// SIMATIC S7-200 SMART project (STEP 7-Micro/WIN SMART), CPU SR40

SYMBOL_TABLE M 符号
急停标志位            M0.0
本地启动标志位          M0.1
远程启动标志位          M0.2
本地停止标志位          M0.3
远程停止标志位          M0.4
主站完成             M1.0
开始读取             M1.1
读取完成1            M1.2
读取完成2            M1.3
读取完成3            M1.4
读取完成4            M1.5
写入完成1            M1.6
写入完成2            M1.7
END_SYMBOL_TABLE

SYMBOL_TABLE 系统符号
Always_On        SM0.0    // 始终接通
First_Scan_On    SM0.1    // 仅在第一个扫描周期时接通
Clock_1s         SM0.5    // 针对 1 s 的周期时间，时钟脉冲接通 0.5 s，断开 0.5 s.
END_SYMBOL_TABLE

SYMBOL_TABLE V 符号
运行指示自动           V10.0
运行指示手动           V10.1
停止指示自动           V10.2
停止指示手动           V10.3
故障指示自动           V10.4
故障指示手动           V10.5
螺杆泵启动自动          V10.6
螺杆泵启动手动          V10.7
罗茨泵启动自动          V11.0
罗茨泵启动手动          V11.1
入口阀自动            V11.2
入口阀手动            V11.3
出口阀自动            V11.4
出口阀手动            V11.5
清洗阀自动            V11.6
清洗阀手动            V11.7
吹扫阀自动            V12.0
吹扫阀手动            V12.1
螺杆泵冷却水阀自动        V12.2
螺杆泵冷却水阀手动        V12.3
罗茨泵冷却水阀自动        V12.4
罗茨泵冷却水阀手动        V12.5
螺杆泵冷却风扇自动        V12.6
螺杆泵冷却风扇手动        V12.7
罗茨泵冷却风扇自动        V13.0
罗茨泵冷却风扇手动        V13.1
排液阀自动            V13.2
排液阀手动            V13.3
罗茨泵启动自动2         V13.4
罗茨泵启动手动2         V13.5
系统故障             V16.0
罗茨泵过载            V16.1
螺杆泵变频器故障报警       V16.2
罗茨泵变频器故障报警       V16.3
冷却水流量低           V16.4
冷却水温度报警          V16.5
冷却水温度停机          V16.6
入口阀打开故障          V16.7
入口阀关闭故障          V17.0
出口阀打开故障          V17.1
出口阀关闭故障          V17.2
螺杆泵冷却风机过载报警      V17.3
罗茨泵冷却风机过载报警      V17.4
螺杆泵维保报警          V17.5
罗茨泵维保报警          V17.6
急停报警             V17.7
罗茨泵变频器故障报警2      V18.0
急停报警2            V18.1
急停报警3            V18.2
运行步              VW20
当前真空度            VD50
当前温度             VD54
排液计时             VW60
清洗计时             VW62
吹扫计时             VW64
冷却水计时            VW66
罗茨泵运行真空度1        VD100
排液间隔时间           VW104
预设清洗时间           VW106
预设吹扫时间           VW108
预设冷却水关闭时间        VW110
螺杆泵手动频率          VW112
罗茨泵手动频率          VW114
螺杆泵停机频率          VW116
冷却水温度报警值         VD118
冷却水温度停机值         VD122
罗茨泵运行真空度2        VD126
罗茨泵停止真空度1        VD130
罗茨泵停止真空度2        VD134
罗茨泵手动频率2         VW138
螺杆泵故障信息          VB200
螺杆泵变频器故障         V201.7
罗茨泵故障信息          VB202
罗茨泵变频器故障         V203.7
罗茨泵故障信息2         VB204
罗茨泵变频器故障2        V205.7
螺杆泵频率电流          VB210
螺杆泵频率            VW210
螺杆泵电流            VW212
罗茨泵频率电流          VB220
罗茨泵频率            VW220
罗茨泵电流            VW222
罗茨泵频率电流2         VB224
罗茨泵频率2           VW224
罗茨泵电流2           VW226
写螺杆泵频率           VB230
螺杆泵频率写入值         VW230
写罗茨泵频率           VB240
罗茨泵频率写入值         VW240
写罗茨泵频率2          VB242
罗茨泵频率写入值2        VW242
中间值1             VD250
中间值2             VD254
螺杆泵当前频率          VD258
中间值3             VD262
中间值4             VD266
螺杆泵当前电流          VD270
中间值5             VD274
中间值6             VD278
罗茨泵当前频率          VD282
中间值7             VD286
中间值8             VD290
罗茨泵当前电流          VD294
写入螺杆泵频率          VW298
写入罗茨泵频率          VW300
写入罗茨泵频率1         VW302
中间值9             VD3000
中间值10            VD3004
中间值11            VD3008
中间值12            VD3012
罗茨泵当前频率2         VD3016
罗茨泵当前电流2         VD3020
写入螺杆泵频率2         VD3024
写入罗茨泵频率2         VD3028
罗茨泵自动频率2         VW3032
中间量13            VW3034
第一页时间1           VW310
第一页时间2           VW312
第一页时间3           VW314
第一页时间4           VW316
第一页时间5           VW318
第一页时间6           VW320
第一页频率1           VW322
第一页频率2           VW324
第一页频率3           VW326
第一页频率4           VW328
第一页频率5           VW330
第一页频率6           VW332
第二页时间1           VW334
第二页时间2           VW336
第二页时间3           VW338
第二页时间4           VW340
第二页时间5           VW342
第二页时间6           VW344
第二页频率1           VW346
第二页频率2           VW348
第二页频率3           VW350
第二页频率4           VW352
第二页频率5           VW354
第二页频率6           VW356
第三页时间1           VW358
第三页时间2           VW360
第三页时间3           VW362
第三页时间4           VW364
第三页时间5           VW366
第三页时间6           VW368
第三页频率1           VW370
第三页频率2           VW372
第三页频率3           VW374
第三页频率4           VW376
第三页频率5           VW378
第三页频率6           VW380
第四页时间1           VW382
第四页时间2           VW384
第四页时间3           VW386
第四页时间4           VW388
第四页时间5           VW390
第四页时间6           VW392
第四页频率1           VW394
第四页频率2           VW396
第四页频率3           VW398
第四页频率4           VW400
第四页频率5           VW402
第四页频率6           VW404
第五页时间1           VW406
第五页时间2           VW408
第五页时间3           VW410
第五页时间4           VW412
第五页时间5           VW414
第五页时间6           VW416
第五页频率1           VW418
第五页频率2           VW420
第五页频率3           VW422
第五页频率4           VW424
第五页频率5           VW426
第五页频率6           VW428
第六页时间1           VW430
第六页时间2           VW432
第六页时间3           VW434
第六页时间4           VW436
第六页时间5           VW438
第六页时间6           VW440
第六页频率1           VW442
第六页频率2           VW444
第六页频率3           VW446
第六页频率4           VW448
第六页频率5           VW450
第六页频率6           VW452
第七页时间1           VW454
第七页时间2           VW456
第七页时间3           VW458
第七页时间4           VW460
第七页时间5           VW462
第七页时间6           VW464
第七页频率1           VW466
第七页频率2           VW468
第七页频率3           VW470
第七页频率4           VW472
第七页频率5           VW474
第七页频率6           VW476
触摸屏页码选择          VW478
实际运行时间1          VW500
实际运行时间2          VW502
实际运行时间3          VW504
实际运行时间4          VW506
实际运行时间5          VW508
实际运行时间6          VW510
实际运行频率1          VW512
实际运行频率2          VW514
实际运行频率3          VW516
实际运行频率4          VW518
实际运行频率5          VW520
实际运行频率6          VW522
step             VW550
螺杆泵自动频率          VW552
罗茨泵自动频率          VW554
螺杆泵运行计时1         VW556
螺杆泵运行计时2         VW558
螺杆泵运行计时3         VW560
螺杆泵运行计时4         VW562
螺杆泵运行计时5         VW564
螺杆泵运行计时6         VW566
中间量9             VW568
螺杆泵总运行时间         VD600
罗茨泵总运行时间         VD604
螺杆泵维保运行时间        VD608
罗茨泵维保运行时间        VD612
螺杆泵维保时间设置        VD616
罗茨泵维保时间设置        VD620
运行时间显示1          VD650    // 螺杆总
运行时间显示2          VD654    // 罗茨总
运行时间显示3          VD658    // 螺杆维保
运行时间显示4          VD662    // 罗茨维保
每秒累加频率1          VD820
每秒累加频率2          VD824
每秒累加频率3          VD828
每秒累加频率4          VD832
每秒累加频率5          VD836
每秒累加频率6          VD840
目标真空度1           VD900
目标真空度2           VD904
目标真空度3           VD908
目标真空度4           VD912
目标真空度5           VD916
目标真空度6           VD920
真空度中间量1          VD924
真空度中间量2          VD928
真空度中间量3          VD932
真空度中间量4          VD936
真空度中间量5          VD940
真空度中间量6          VD944
END_SYMBOL_TABLE

ORGANIZATION_BLOCK MAIN:OB1
TITLE=程序注释
BEGIN
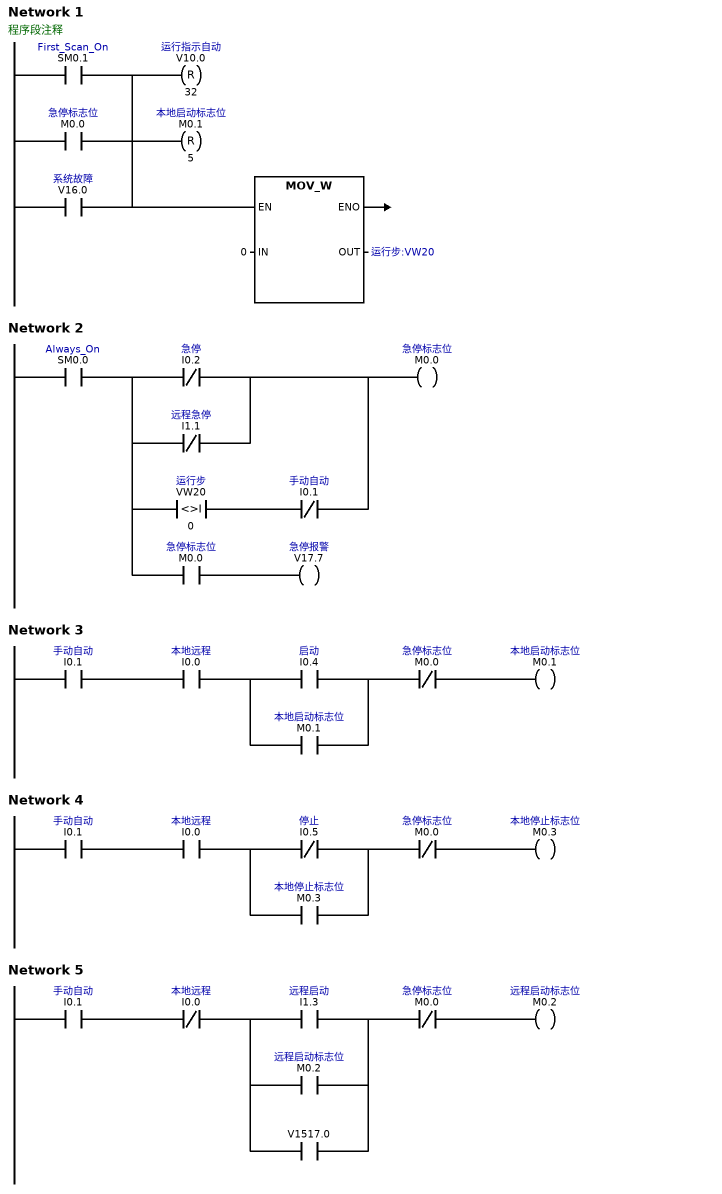
Network 1
// 程序段注释
LD     First_Scan_On:SM0.1
O      急停标志位:M0.0
O      系统故障:V16.0
R      运行指示自动:V10.0, 32
R      本地启动标志位:M0.1, 5
MOVW   0, 运行步:VW20
Network 2
LD     Always_On:SM0.0
LPS
LDN    急停:I0.2
ON     远程急停:I1.1
LDW<>  运行步:VW20, 0
AN     手动自动:I0.1
OLD
ALD
=      急停标志位:M0.0
LPP
A      急停标志位:M0.0
=      急停报警:V17.7
Network 3
LD     手动自动:I0.1
A      本地远程:I0.0
LD     启动:I0.4
O      本地启动标志位:M0.1
ALD
AN     急停标志位:M0.0
=      本地启动标志位:M0.1
Network 4
LD     手动自动:I0.1
A      本地远程:I0.0
LDN    停止:I0.5
O      本地停止标志位:M0.3
ALD
AN     急停标志位:M0.0
=      本地停止标志位:M0.3
Network 5
LD     手动自动:I0.1
AN     本地远程:I0.0
LD     远程启动:I1.3
O      远程启动标志位:M0.2
O      V1517.0
ALD
AN     急停标志位:M0.0
=      远程启动标志位:M0.2
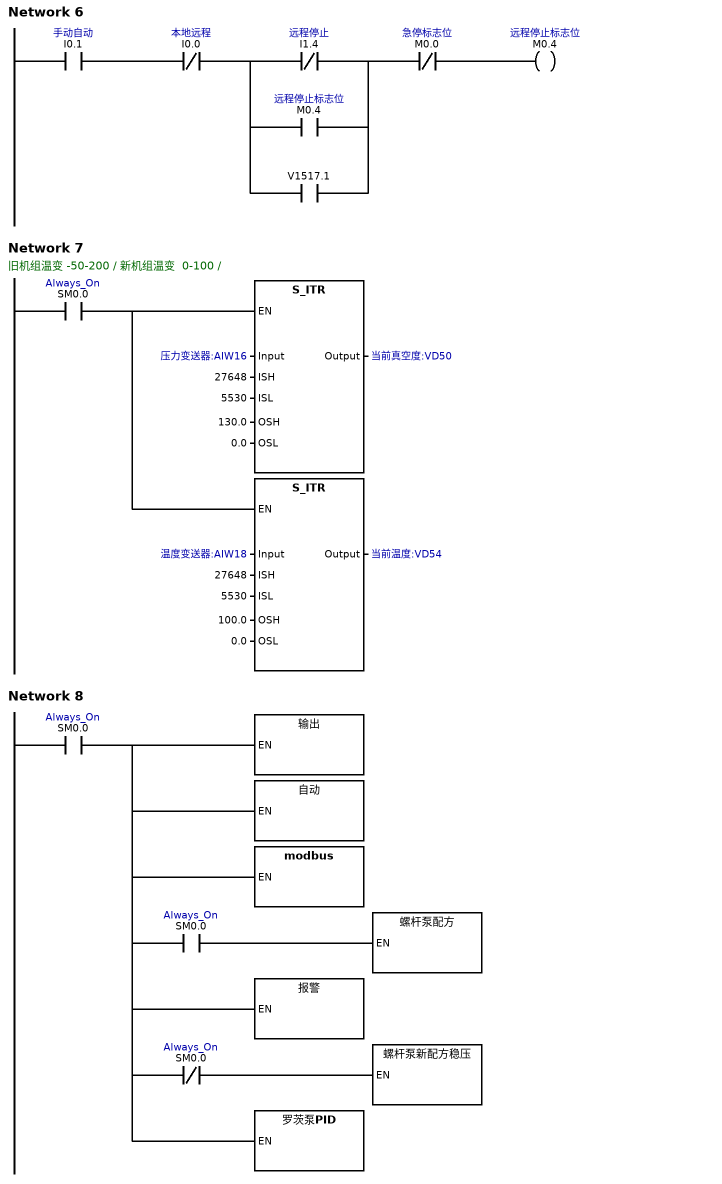
Network 6
LD     手动自动:I0.1
AN     本地远程:I0.0
LDN    远程停止:I1.4
O      远程停止标志位:M0.4
O      V1517.1
ALD
AN     急停标志位:M0.0
=      远程停止标志位:M0.4
Network 7
// 旧机组温变 -50-200
// 新机组温变  0-100
// 
LD     Always_On:SM0.0
CALL   S_ITR:SBR1, 压力变送器:AIW16, 27648, 5530, 130.0, 0.0, 当前真空度:VD50
CALL   S_ITR:SBR1, 温度变送器:AIW18, 27648, 5530, 100.0, 0.0, 当前温度:VD54
Network 8
LD     Always_On:SM0.0
LPS
CALL   输出:SBR0
CALL   自动:SBR2
CALL   modbus:SBR3
A      Always_On:SM0.0
CALL   螺杆泵配方:SBR4
LRD
CALL   报警:SBR6
LRD
AN     Always_On:SM0.0
CALL   螺杆泵新配方稳压:SBR15
LPP
CALL   罗茨泵PID:SBR5
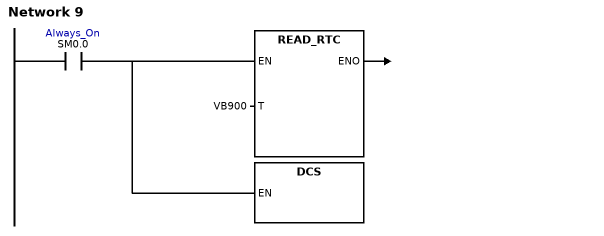
Network 9
LD     Always_On:SM0.0
TODR   VB900
CALL   DCS:SBR11
END_ORGANIZATION_BLOCK

SUBROUTINE_BLOCK 输出:SBR0
TITLE=子程序注释
BEGIN
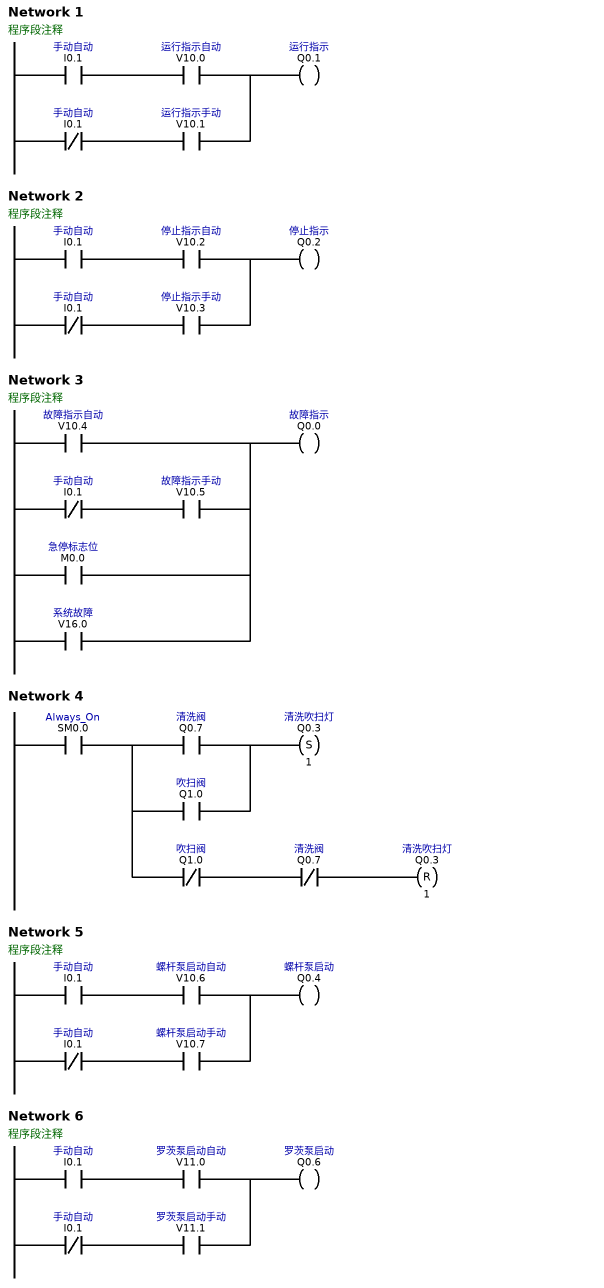
Network 1
// 程序段注释
LD     手动自动:I0.1
A      运行指示自动:V10.0
LDN    手动自动:I0.1
A      运行指示手动:V10.1
OLD
=      运行指示:Q0.1
Network 2
// 程序段注释
LD     手动自动:I0.1
A      停止指示自动:V10.2
LDN    手动自动:I0.1
A      停止指示手动:V10.3
OLD
=      停止指示:Q0.2
Network 3
// 程序段注释
LD     故障指示自动:V10.4
LDN    手动自动:I0.1
A      故障指示手动:V10.5
OLD
O      急停标志位:M0.0
O      系统故障:V16.0
=      故障指示:Q0.0
Network 4
LD     Always_On:SM0.0
LPS
LD     清洗阀:Q0.7
O      吹扫阀:Q1.0
ALD
S      清洗吹扫灯:Q0.3, 1
LPP
AN     吹扫阀:Q1.0
AN     清洗阀:Q0.7
R      清洗吹扫灯:Q0.3, 1
Network 5
// 程序段注释
LD     手动自动:I0.1
A      螺杆泵启动自动:V10.6
LDN    手动自动:I0.1
A      螺杆泵启动手动:V10.7
OLD
=      螺杆泵启动:Q0.4
Network 6
// 程序段注释
LD     手动自动:I0.1
A      罗茨泵启动自动:V11.0
LDN    手动自动:I0.1
A      罗茨泵启动手动:V11.1
OLD
=      罗茨泵启动:Q0.6
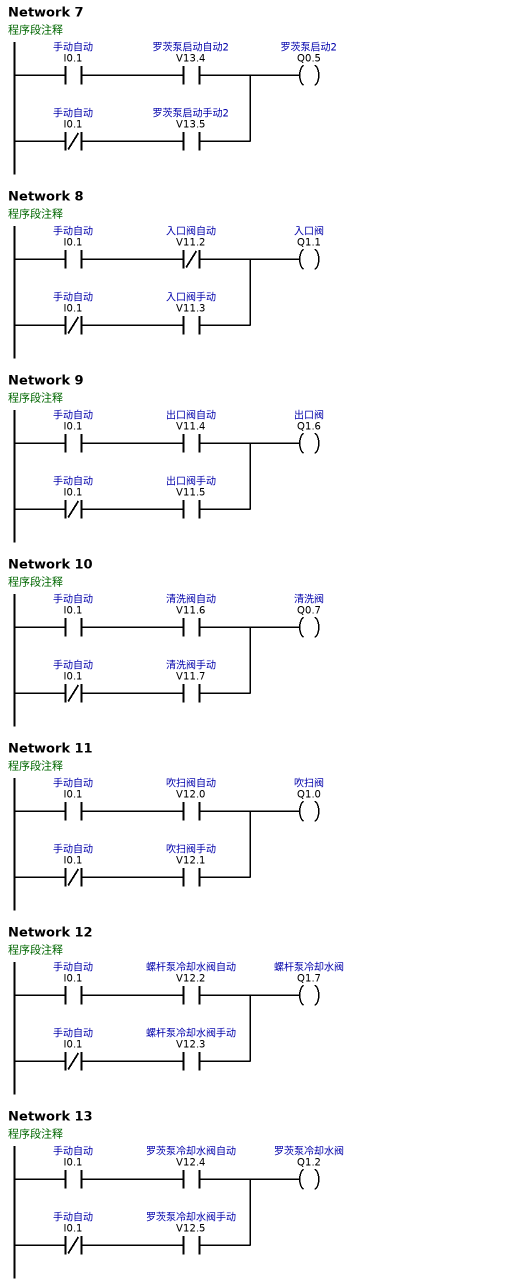
Network 7
// 程序段注释
LD     手动自动:I0.1
A      罗茨泵启动自动2:V13.4
LDN    手动自动:I0.1
A      罗茨泵启动手动2:V13.5
OLD
=      罗茨泵启动2:Q0.5
Network 8
// 程序段注释
LD     手动自动:I0.1
AN     入口阀自动:V11.2
LDN    手动自动:I0.1
A      入口阀手动:V11.3
OLD
=      入口阀:Q1.1
Network 9
// 程序段注释
LD     手动自动:I0.1
A      出口阀自动:V11.4
LDN    手动自动:I0.1
A      出口阀手动:V11.5
OLD
=      出口阀:Q1.6
Network 10
// 程序段注释
LD     手动自动:I0.1
A      清洗阀自动:V11.6
LDN    手动自动:I0.1
A      清洗阀手动:V11.7
OLD
=      清洗阀:Q0.7
Network 11
// 程序段注释
LD     手动自动:I0.1
A      吹扫阀自动:V12.0
LDN    手动自动:I0.1
A      吹扫阀手动:V12.1
OLD
=      吹扫阀:Q1.0
Network 12
// 程序段注释
LD     手动自动:I0.1
A      螺杆泵冷却水阀自动:V12.2
LDN    手动自动:I0.1
A      螺杆泵冷却水阀手动:V12.3
OLD
=      螺杆泵冷却水阀:Q1.7
Network 13
// 程序段注释
LD     手动自动:I0.1
A      罗茨泵冷却水阀自动:V12.4
LDN    手动自动:I0.1
A      罗茨泵冷却水阀手动:V12.5
OLD
=      罗茨泵冷却水阀:Q1.2
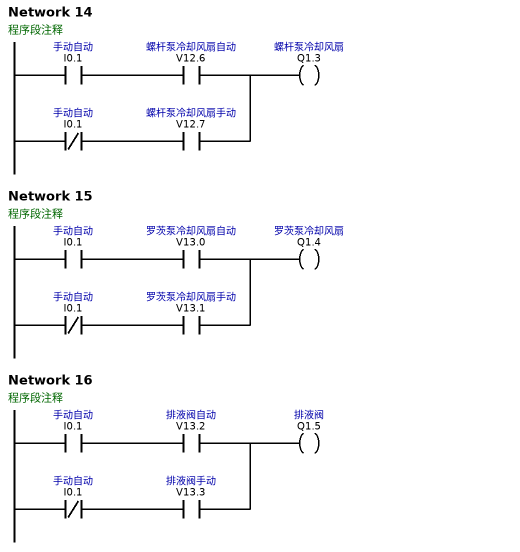
Network 14
// 程序段注释
LD     手动自动:I0.1
A      螺杆泵冷却风扇自动:V12.6
LDN    手动自动:I0.1
A      螺杆泵冷却风扇手动:V12.7
OLD
=      螺杆泵冷却风扇:Q1.3
Network 15
// 程序段注释
LD     手动自动:I0.1
A      罗茨泵冷却风扇自动:V13.0
LDN    手动自动:I0.1
A      罗茨泵冷却风扇手动:V13.1
OLD
=      罗茨泵冷却风扇:Q1.4
Network 16
// 程序段注释
LD     手动自动:I0.1
A      排液阀自动:V13.2
LDN    手动自动:I0.1
A      排液阀手动:V13.3
OLD
=      排液阀:Q1.5
END_SUBROUTINE_BLOCK

// SBR1: protected block, not included

SUBROUTINE_BLOCK 自动:SBR2
TITLE=子程序注释
BEGIN
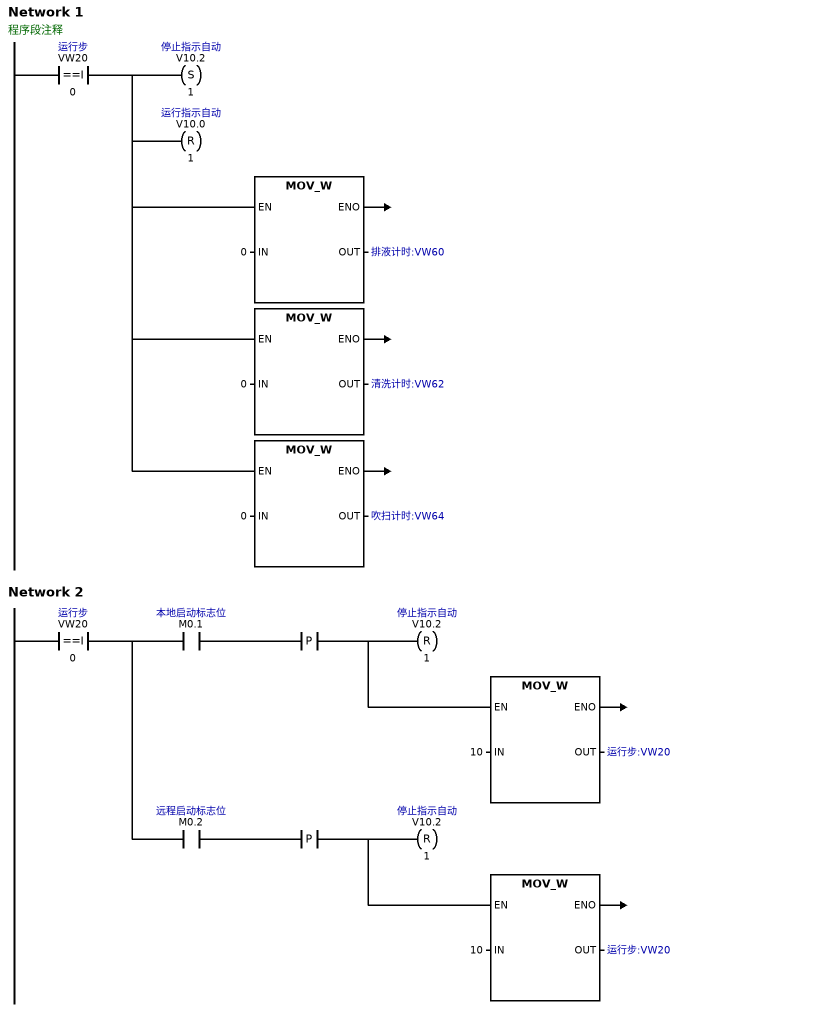
Network 1
// 程序段注释
LDW=   运行步:VW20, 0
S      停止指示自动:V10.2, 1
R      运行指示自动:V10.0, 1
MOVW   0, 排液计时:VW60
MOVW   0, 清洗计时:VW62
MOVW   0, 吹扫计时:VW64
Network 2
LDW=   运行步:VW20, 0
LPS
A      本地启动标志位:M0.1
EU
R      停止指示自动:V10.2, 1
MOVW   10, 运行步:VW20
LPP
A      远程启动标志位:M0.2
EU
R      停止指示自动:V10.2, 1
MOVW   10, 运行步:VW20
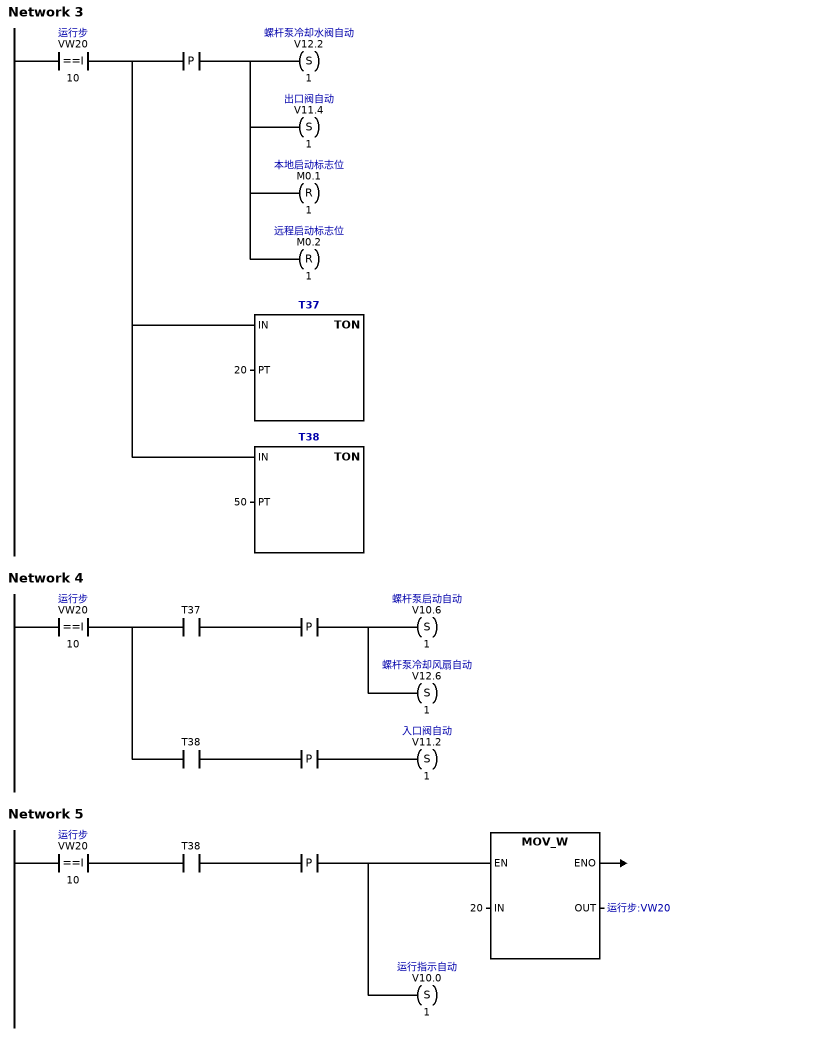
Network 3
LDW=   运行步:VW20, 10
LPS
EU
S      螺杆泵冷却水阀自动:V12.2, 1
S      出口阀自动:V11.4, 1
R      本地启动标志位:M0.1, 1
R      远程启动标志位:M0.2, 1
LPP
TON    T37, 20
TON    T38, 50
Network 4
LDW=   运行步:VW20, 10
LPS
A      T37
EU
S      螺杆泵启动自动:V10.6, 1
S      螺杆泵冷却风扇自动:V12.6, 1
LPP
A      T38
EU
S      入口阀自动:V11.2, 1
Network 5
LDW=   运行步:VW20, 10
A      T38
EU
MOVW   20, 运行步:VW20
S      运行指示自动:V10.0, 1
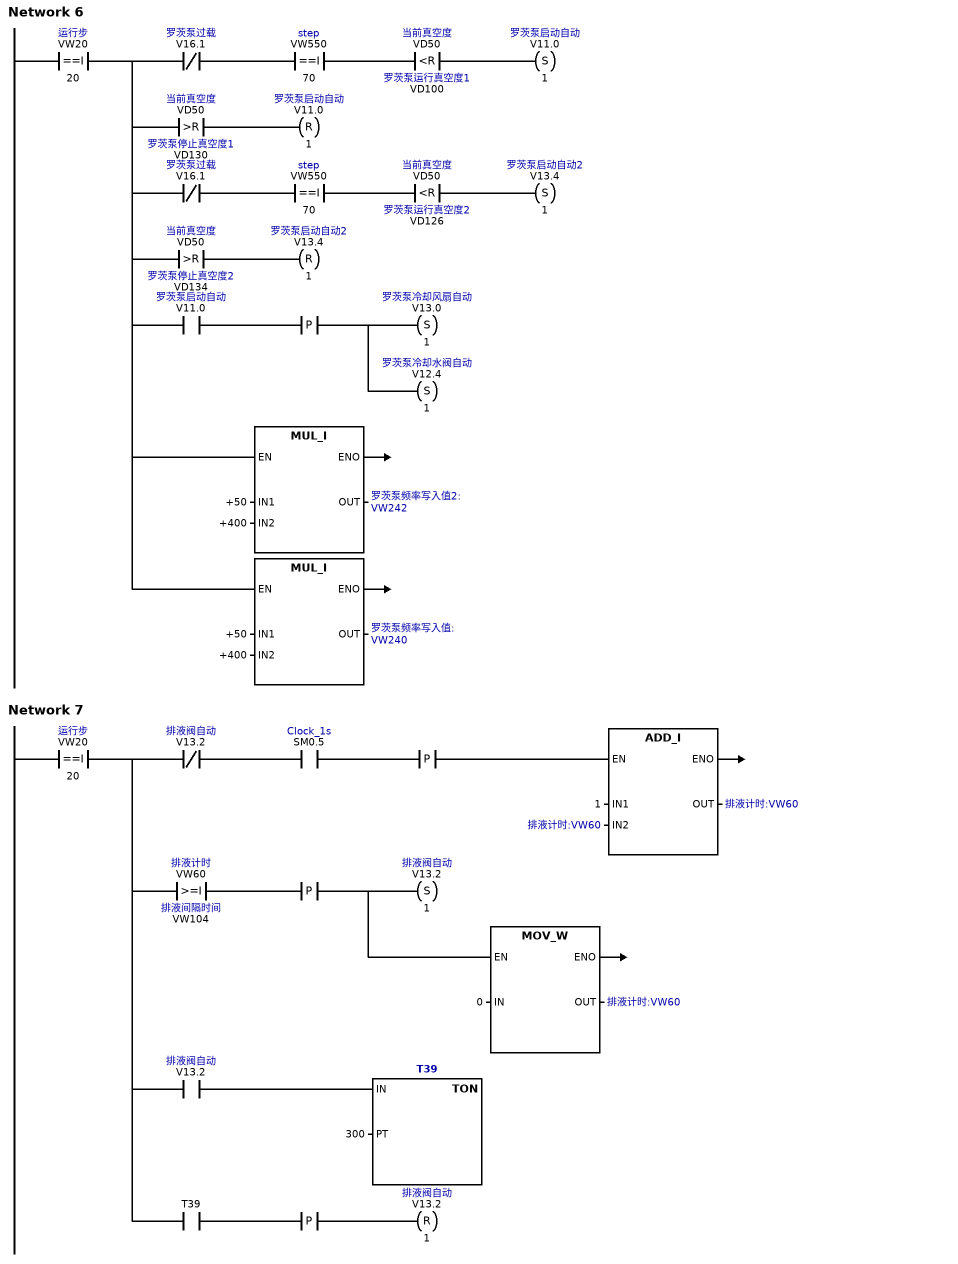
Network 6
LDW=   运行步:VW20, 20
LPS
AN     罗茨泵过载:V16.1
AW=    step:VW550, 70
AR<    当前真空度:VD50, 罗茨泵运行真空度1:VD100
S      罗茨泵启动自动:V11.0, 1
LRD
AR>    当前真空度:VD50, 罗茨泵停止真空度1:VD130
R      罗茨泵启动自动:V11.0, 1
LRD
AN     罗茨泵过载:V16.1
AW=    step:VW550, 70
AR<    当前真空度:VD50, 罗茨泵运行真空度2:VD126
S      罗茨泵启动自动2:V13.4, 1
LRD
AR>    当前真空度:VD50, 罗茨泵停止真空度2:VD134
R      罗茨泵启动自动2:V13.4, 1
LRD
A      罗茨泵启动自动:V11.0
EU
S      罗茨泵冷却风扇自动:V13.0, 1
S      罗茨泵冷却水阀自动:V12.4, 1
LPP
MOVW   +50, 罗茨泵频率写入值2:VW242
*I     +400, 罗茨泵频率写入值2:VW242
MOVW   +50, 罗茨泵频率写入值:VW240
*I     +400, 罗茨泵频率写入值:VW240
Network 7
LDW=   运行步:VW20, 20
LPS
AN     排液阀自动:V13.2
A      Clock_1s:SM0.5
EU
+I     1, 排液计时:VW60
LRD
AW>=   排液计时:VW60, 排液间隔时间:VW104
EU
S      排液阀自动:V13.2, 1
MOVW   0, 排液计时:VW60
LPP
LPS
A      排液阀自动:V13.2
TON    T39, 300
LPP
A      T39
EU
R      排液阀自动:V13.2, 1
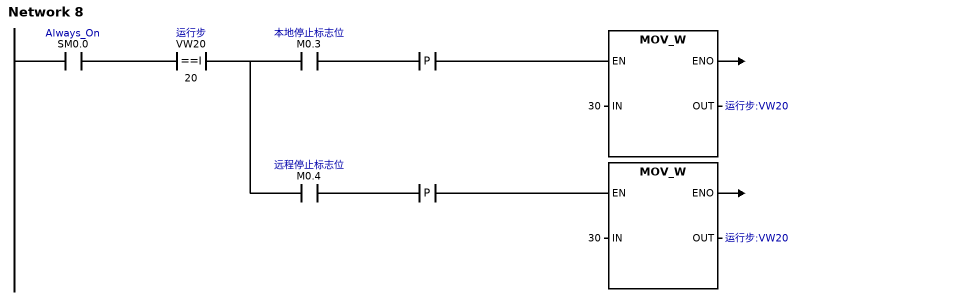
Network 8
LD     Always_On:SM0.0
AW=    运行步:VW20, 20
LPS
A      本地停止标志位:M0.3
EU
MOVW   30, 运行步:VW20
LPP
A      远程停止标志位:M0.4
EU
MOVW   30, 运行步:VW20
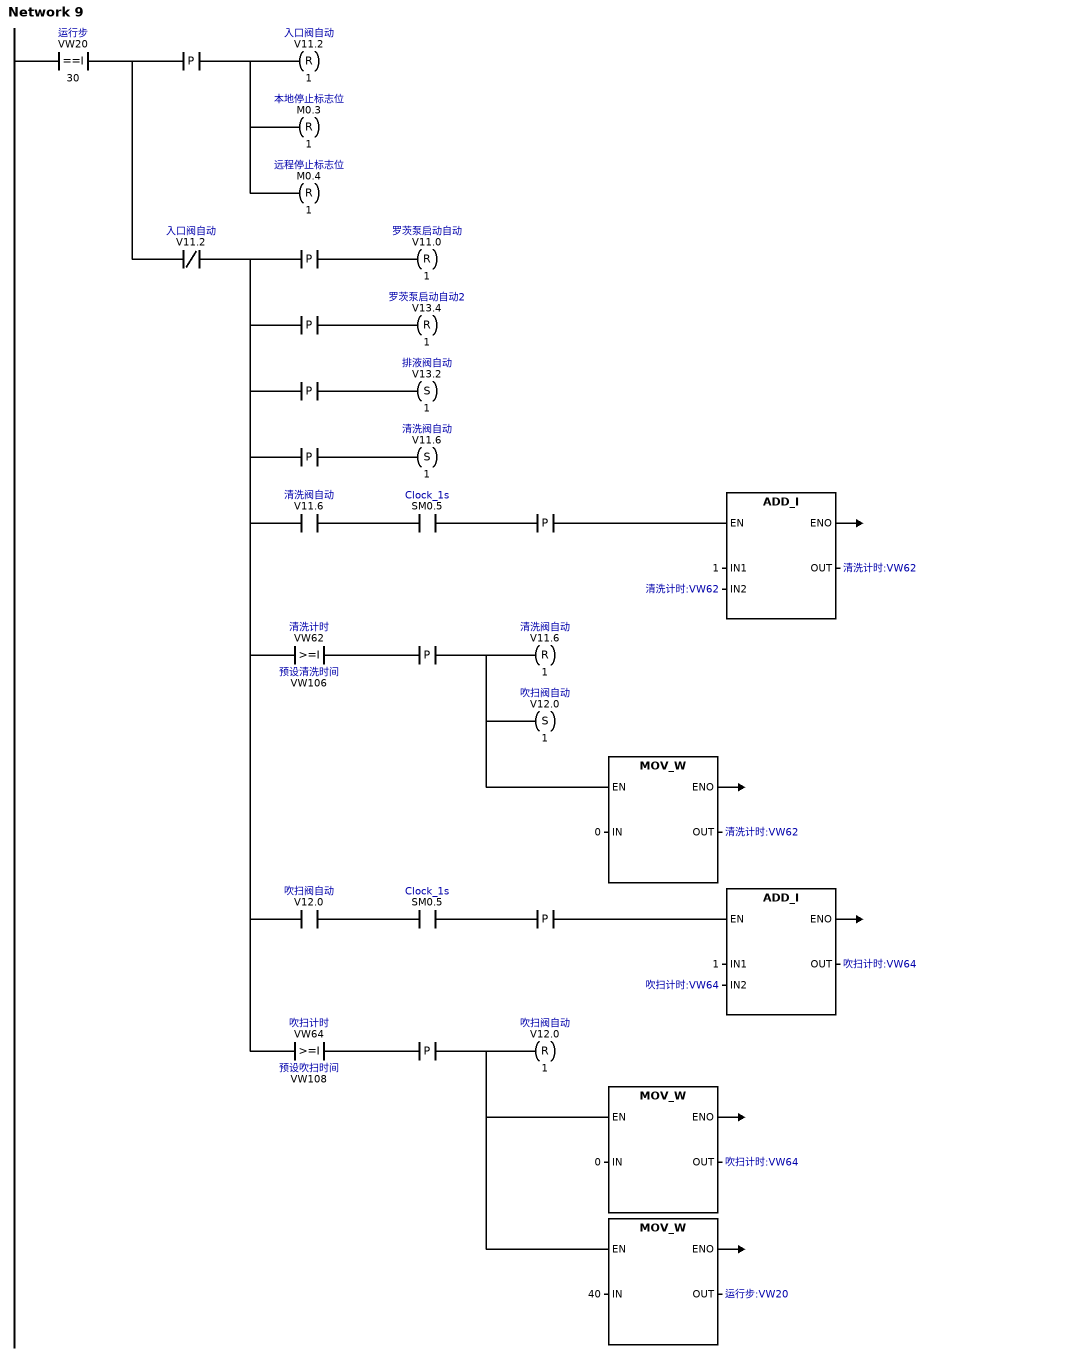
Network 9
LDW=   运行步:VW20, 30
LPS
EU
R      入口阀自动:V11.2, 1
R      本地停止标志位:M0.3, 1
R      远程停止标志位:M0.4, 1
LPP
AN     入口阀自动:V11.2
LPS
EU
R      罗茨泵启动自动:V11.0, 1
LRD
EU
R      罗茨泵启动自动2:V13.4, 1
LRD
EU
S      排液阀自动:V13.2, 1
LRD
EU
S      清洗阀自动:V11.6, 1
LRD
A      清洗阀自动:V11.6
A      Clock_1s:SM0.5
EU
+I     1, 清洗计时:VW62
LRD
AW>=   清洗计时:VW62, 预设清洗时间:VW106
EU
R      清洗阀自动:V11.6, 1
S      吹扫阀自动:V12.0, 1
MOVW   0, 清洗计时:VW62
LRD
A      吹扫阀自动:V12.0
A      Clock_1s:SM0.5
EU
+I     1, 吹扫计时:VW64
LPP
AW>=   吹扫计时:VW64, 预设吹扫时间:VW108
EU
R      吹扫阀自动:V12.0, 1
MOVW   0, 吹扫计时:VW64
MOVW   40, 运行步:VW20
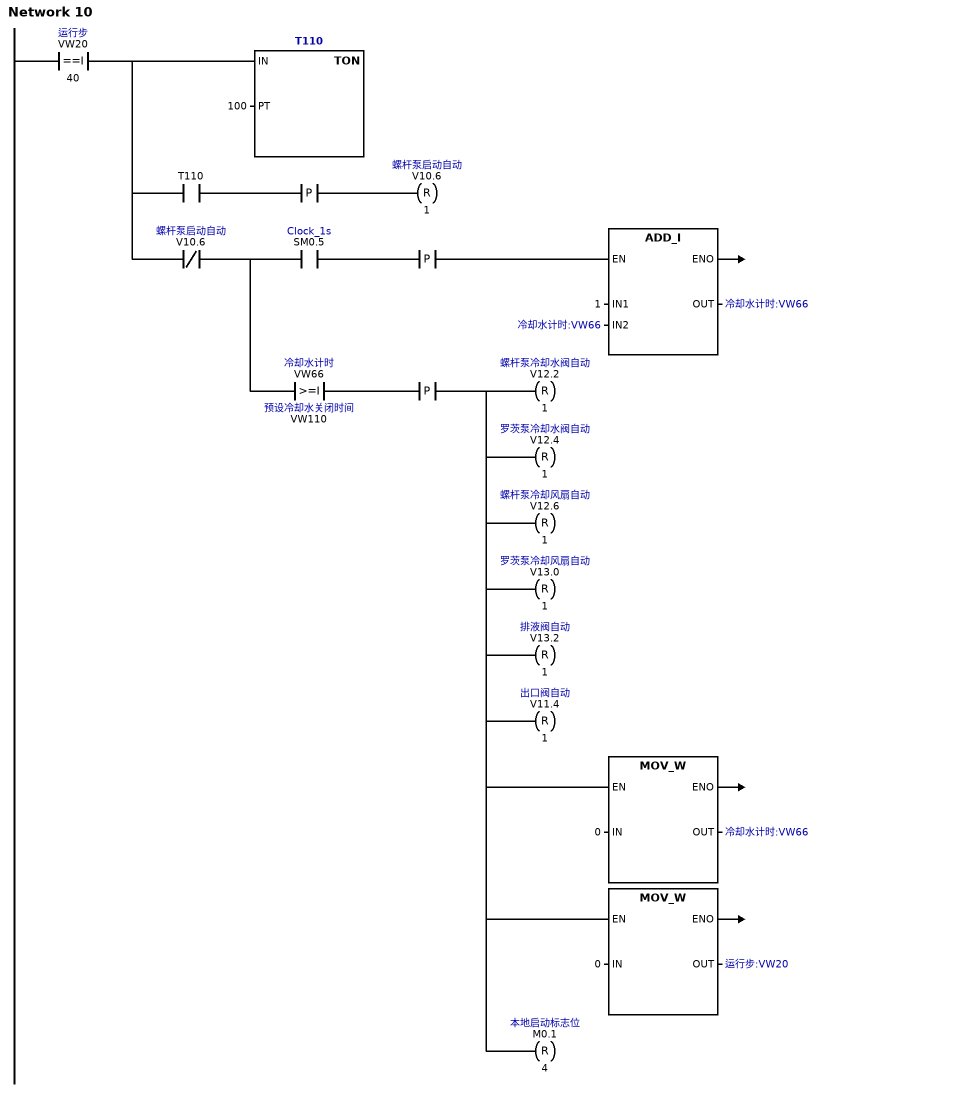
Network 10
LDW=   运行步:VW20, 40
LPS
TON    T110, 100
A      T110
EU
R      螺杆泵启动自动:V10.6, 1
LPP
AN     螺杆泵启动自动:V10.6
LPS
A      Clock_1s:SM0.5
EU
+I     1, 冷却水计时:VW66
LPP
AW>=   冷却水计时:VW66, 预设冷却水关闭时间:VW110
EU
R      螺杆泵冷却水阀自动:V12.2, 1
R      罗茨泵冷却水阀自动:V12.4, 1
R      螺杆泵冷却风扇自动:V12.6, 1
R      罗茨泵冷却风扇自动:V13.0, 1
R      排液阀自动:V13.2, 1
R      出口阀自动:V11.4, 1
MOVW   0, 冷却水计时:VW66
MOVW   0, 运行步:VW20
R      本地启动标志位:M0.1, 4
END_SUBROUTINE_BLOCK

SUBROUTINE_BLOCK modbus:SBR3
TITLE=子程序注释
BEGIN
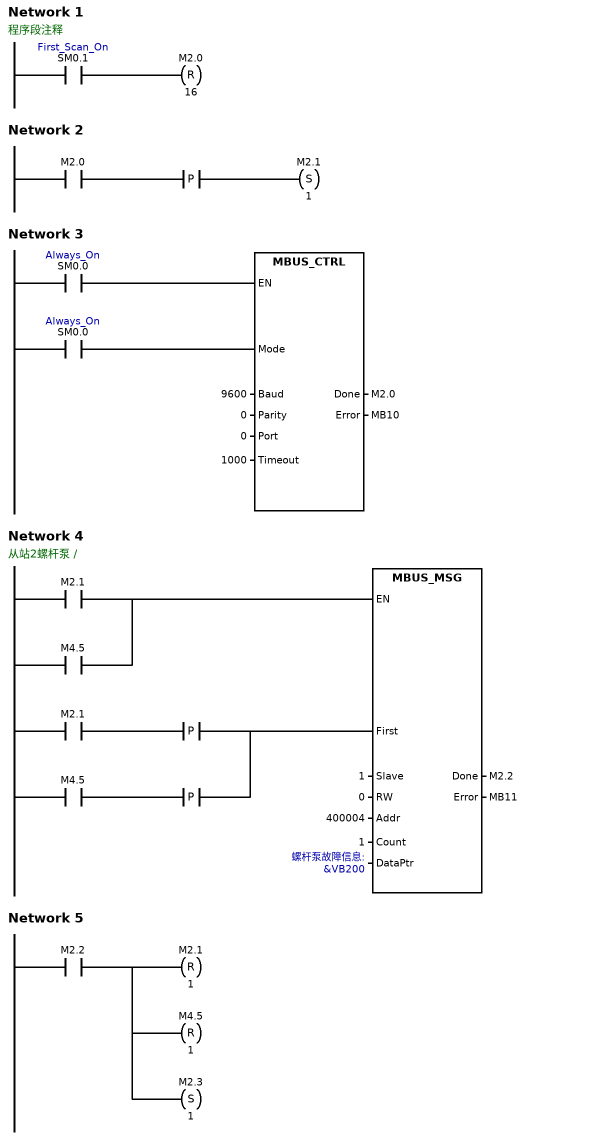
Network 1
// 程序段注释
LD     First_Scan_On:SM0.1
R      M2.0, 16
Network 2
LD     M2.0
EU
S      M2.1, 1
Network 3
LD     Always_On:SM0.0
=      L60.0
LD     Always_On:SM0.0
=      L63.7
LD     L60.0
CALL   MBUS_CTRL:SBR7, L63.7, 9600, 0, 0, 1000, M2.0, MB10
Network 4
// 从站2螺杆泵
// 
LD     M2.1
O      M4.5
=      L60.0
LD     M2.1
EU
LD     M4.5
EU
OLD
=      L63.7
LD     L60.0
CALL   MBUS_MSG:SBR8, L63.7, 1, 0, 400004, 1, &螺杆泵故障信息:VB200, M2.2, MB11
Network 5
LD     M2.2
R      M2.1, 1
R      M4.5, 1
S      M2.3, 1
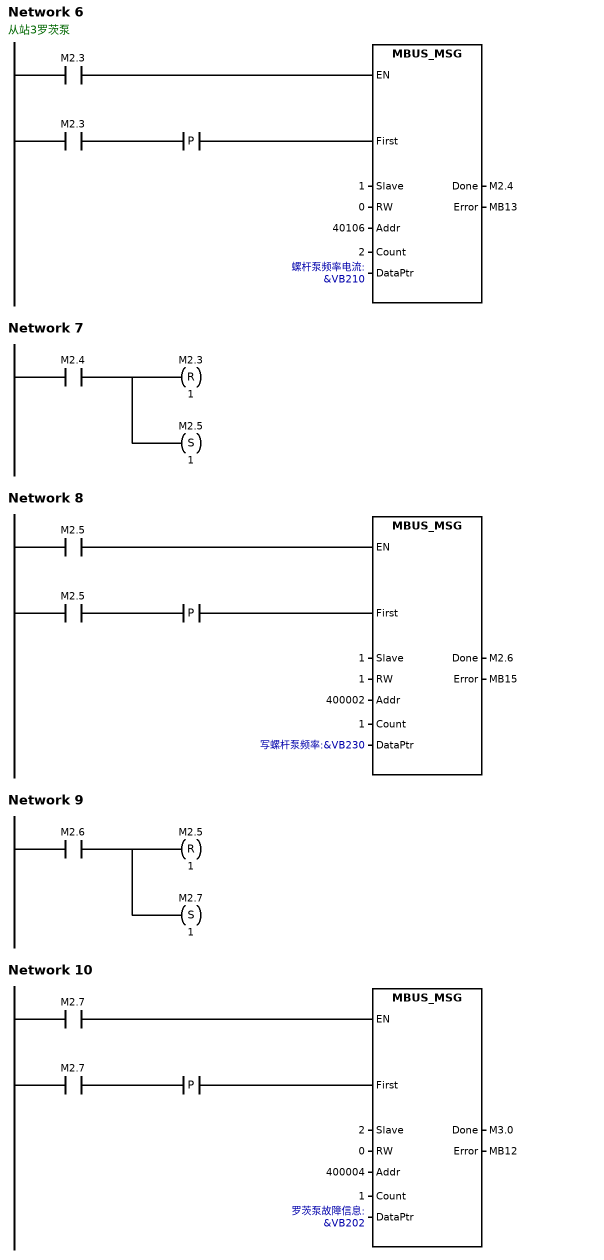
Network 6
// 从站3罗茨泵
LD     M2.3
=      L60.0
LD     M2.3
EU
=      L63.7
LD     L60.0
CALL   MBUS_MSG:SBR8, L63.7, 1, 0, 40106, 2, &螺杆泵频率电流:VB210, M2.4, MB13
Network 7
LD     M2.4
R      M2.3, 1
S      M2.5, 1
Network 8
LD     M2.5
=      L60.0
LD     M2.5
EU
=      L63.7
LD     L60.0
CALL   MBUS_MSG:SBR8, L63.7, 1, 1, 400002, 1, &写螺杆泵频率:VB230, M2.6, MB15
Network 9
LD     M2.6
R      M2.5, 1
S      M2.7, 1
Network 10
LD     M2.7
=      L60.0
LD     M2.7
EU
=      L63.7
LD     L60.0
CALL   MBUS_MSG:SBR8, L63.7, 2, 0, 400004, 1, &罗茨泵故障信息:VB202, M3.0, MB12
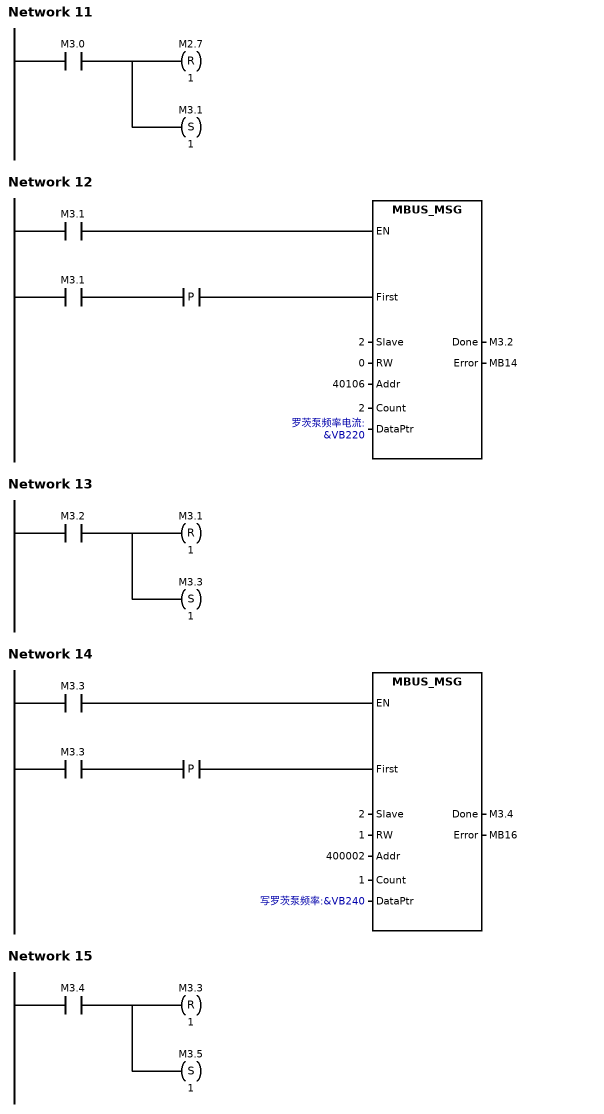
Network 11
LD     M3.0
R      M2.7, 1
S      M3.1, 1
Network 12
LD     M3.1
=      L60.0
LD     M3.1
EU
=      L63.7
LD     L60.0
CALL   MBUS_MSG:SBR8, L63.7, 2, 0, 40106, 2, &罗茨泵频率电流:VB220, M3.2, MB14
Network 13
LD     M3.2
R      M3.1, 1
S      M3.3, 1
Network 14
LD     M3.3
=      L60.0
LD     M3.3
EU
=      L63.7
LD     L60.0
CALL   MBUS_MSG:SBR8, L63.7, 2, 1, 400002, 1, &写罗茨泵频率:VB240, M3.4, MB16
Network 15
LD     M3.4
R      M3.3, 1
S      M3.5, 1
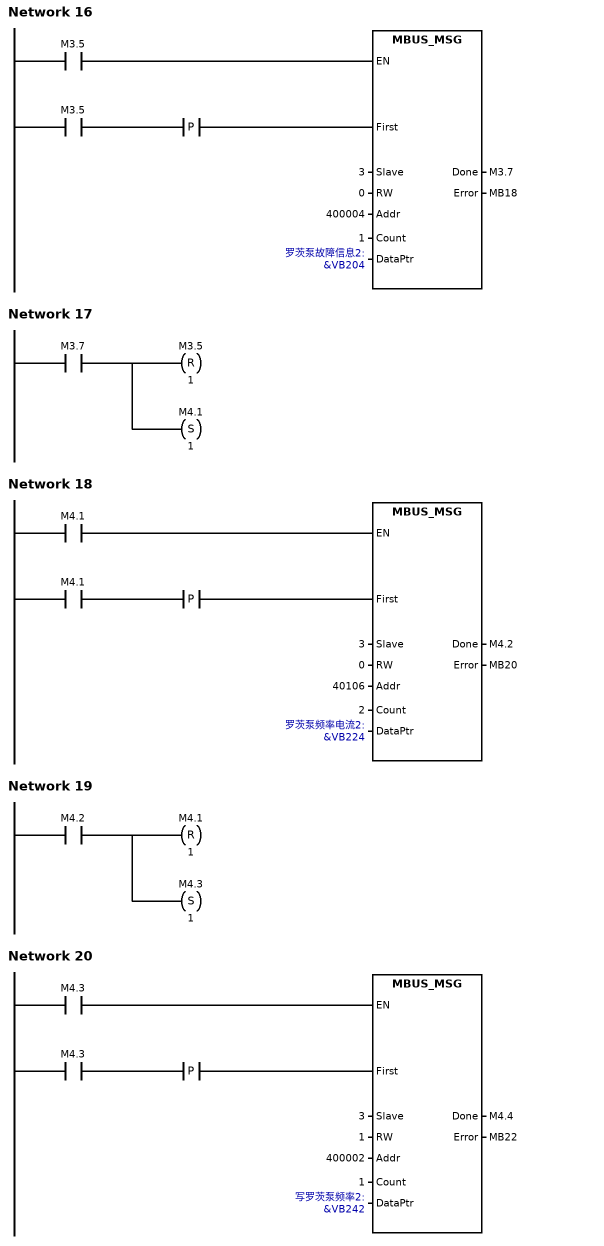
Network 16
LD     M3.5
=      L60.0
LD     M3.5
EU
=      L63.7
LD     L60.0
CALL   MBUS_MSG:SBR8, L63.7, 3, 0, 400004, 1, &罗茨泵故障信息2:VB204, M3.7, MB18
Network 17
LD     M3.7
R      M3.5, 1
S      M4.1, 1
Network 18
LD     M4.1
=      L60.0
LD     M4.1
EU
=      L63.7
LD     L60.0
CALL   MBUS_MSG:SBR8, L63.7, 3, 0, 40106, 2, &罗茨泵频率电流2:VB224, M4.2, MB20
Network 19
LD     M4.2
R      M4.1, 1
S      M4.3, 1
Network 20
LD     M4.3
=      L60.0
LD     M4.3
EU
=      L63.7
LD     L60.0
CALL   MBUS_MSG:SBR8, L63.7, 3, 1, 400002, 1, &写罗茨泵频率2:VB242, M4.4, MB22
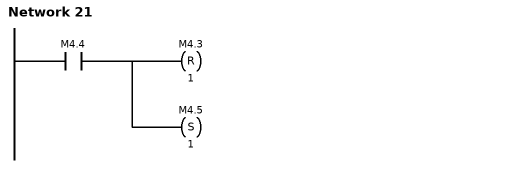
Network 21
LD     M4.4
R      M4.3, 1
S      M4.5, 1
END_SUBROUTINE_BLOCK

SUBROUTINE_BLOCK 螺杆泵配方:SBR4
TITLE=子程序注释
BEGIN
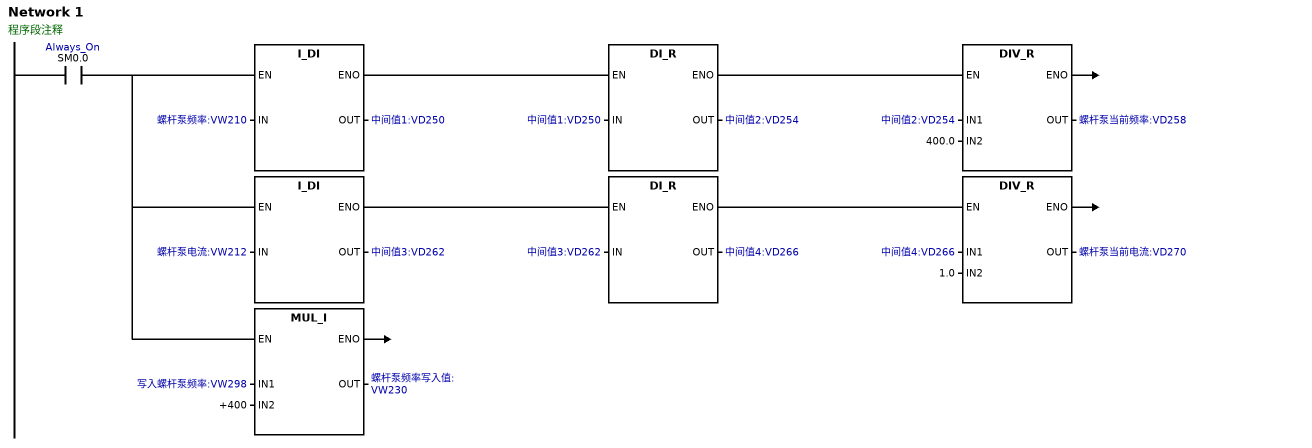
Network 1
// 程序段注释
LD     Always_On:SM0.0
LPS
ITD    螺杆泵频率:VW210, 中间值1:VD250
AENO
DTR    中间值1:VD250, 中间值2:VD254
AENO
MOVR   中间值2:VD254, 螺杆泵当前频率:VD258
/R     400.0, 螺杆泵当前频率:VD258
LRD
ITD    螺杆泵电流:VW212, 中间值3:VD262
AENO
DTR    中间值3:VD262, 中间值4:VD266
AENO
MOVR   中间值4:VD266, 螺杆泵当前电流:VD270
/R     1.0, 螺杆泵当前电流:VD270
LPP
MOVW   写入螺杆泵频率:VW298, 螺杆泵频率写入值:VW230
*I     +400, 螺杆泵频率写入值:VW230
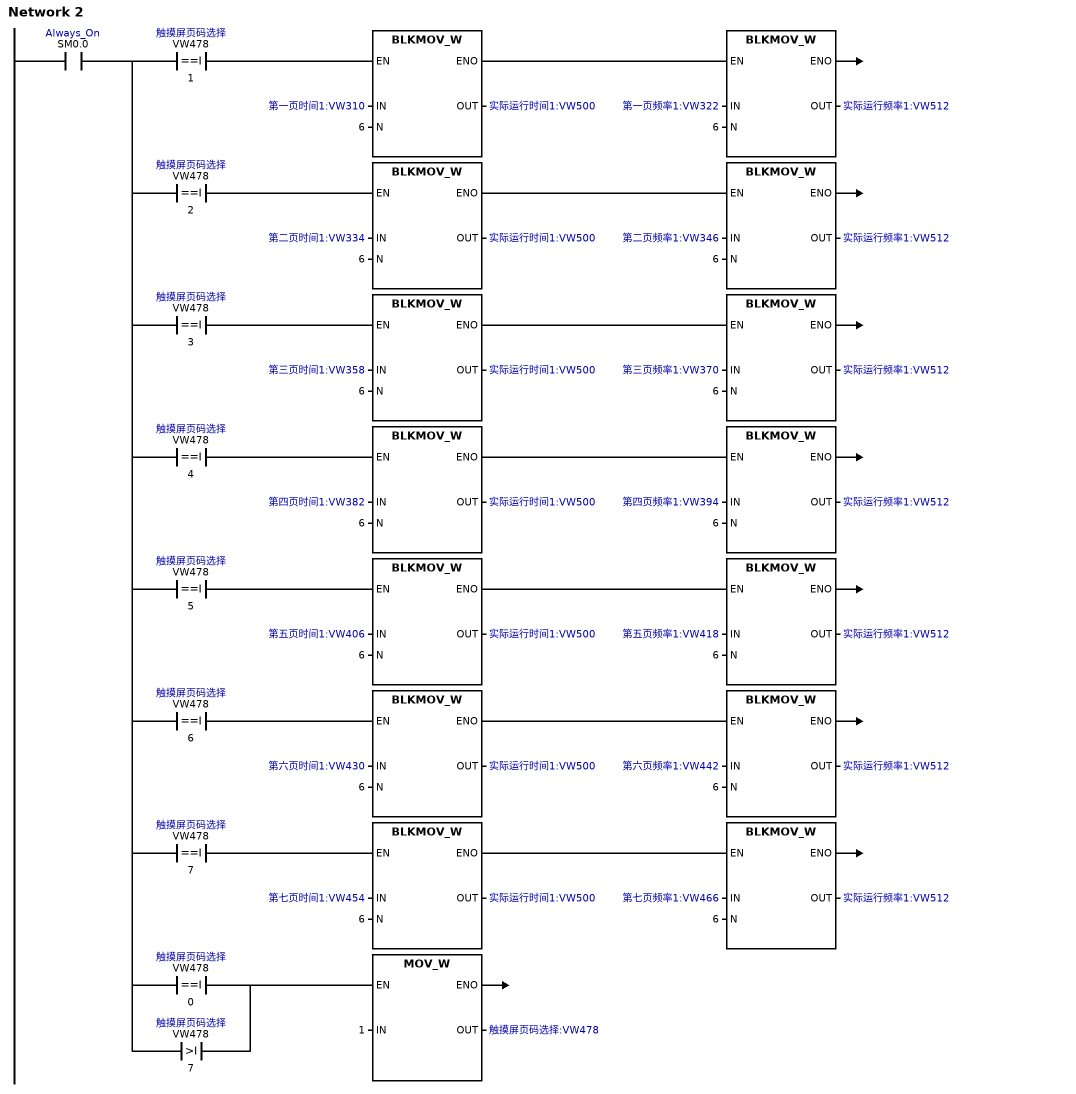
Network 2
LD     Always_On:SM0.0
LPS
AW=    触摸屏页码选择:VW478, 1
BMW    第一页时间1:VW310, 实际运行时间1:VW500, 6
AENO
BMW    第一页频率1:VW322, 实际运行频率1:VW512, 6
LRD
AW=    触摸屏页码选择:VW478, 2
BMW    第二页时间1:VW334, 实际运行时间1:VW500, 6
AENO
BMW    第二页频率1:VW346, 实际运行频率1:VW512, 6
LRD
AW=    触摸屏页码选择:VW478, 3
BMW    第三页时间1:VW358, 实际运行时间1:VW500, 6
AENO
BMW    第三页频率1:VW370, 实际运行频率1:VW512, 6
LRD
AW=    触摸屏页码选择:VW478, 4
BMW    第四页时间1:VW382, 实际运行时间1:VW500, 6
AENO
BMW    第四页频率1:VW394, 实际运行频率1:VW512, 6
LRD
AW=    触摸屏页码选择:VW478, 5
BMW    第五页时间1:VW406, 实际运行时间1:VW500, 6
AENO
BMW    第五页频率1:VW418, 实际运行频率1:VW512, 6
LRD
AW=    触摸屏页码选择:VW478, 6
BMW    第六页时间1:VW430, 实际运行时间1:VW500, 6
AENO
BMW    第六页频率1:VW442, 实际运行频率1:VW512, 6
LRD
AW=    触摸屏页码选择:VW478, 7
BMW    第七页时间1:VW454, 实际运行时间1:VW500, 6
AENO
BMW    第七页频率1:VW466, 实际运行频率1:VW512, 6
LPP
LDW=   触摸屏页码选择:VW478, 0
OW>    触摸屏页码选择:VW478, 7
ALD
MOVW   1, 触摸屏页码选择:VW478
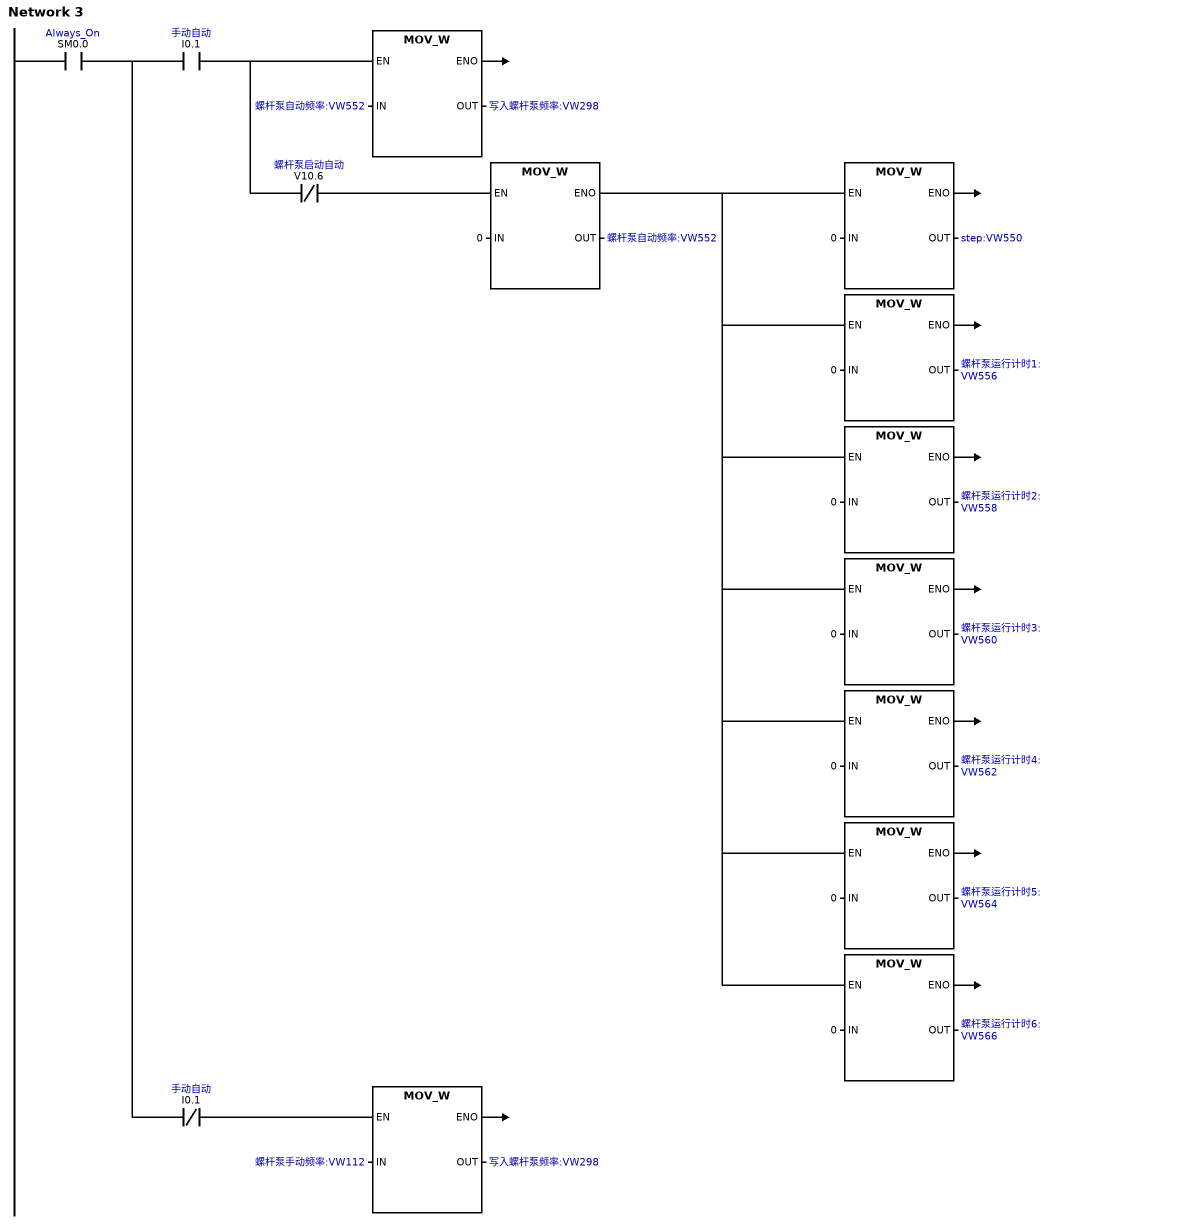
Network 3
LD     Always_On:SM0.0
LPS
A      手动自动:I0.1
MOVW   螺杆泵自动频率:VW552, 写入螺杆泵频率:VW298
AN     螺杆泵启动自动:V10.6
MOVW   0, 螺杆泵自动频率:VW552
AENO
MOVW   0, step:VW550
MOVW   0, 螺杆泵运行计时1:VW556
MOVW   0, 螺杆泵运行计时2:VW558
MOVW   0, 螺杆泵运行计时3:VW560
MOVW   0, 螺杆泵运行计时4:VW562
MOVW   0, 螺杆泵运行计时5:VW564
MOVW   0, 螺杆泵运行计时6:VW566
LPP
AN     手动自动:I0.1
MOVW   螺杆泵手动频率:VW112, 写入螺杆泵频率:VW298
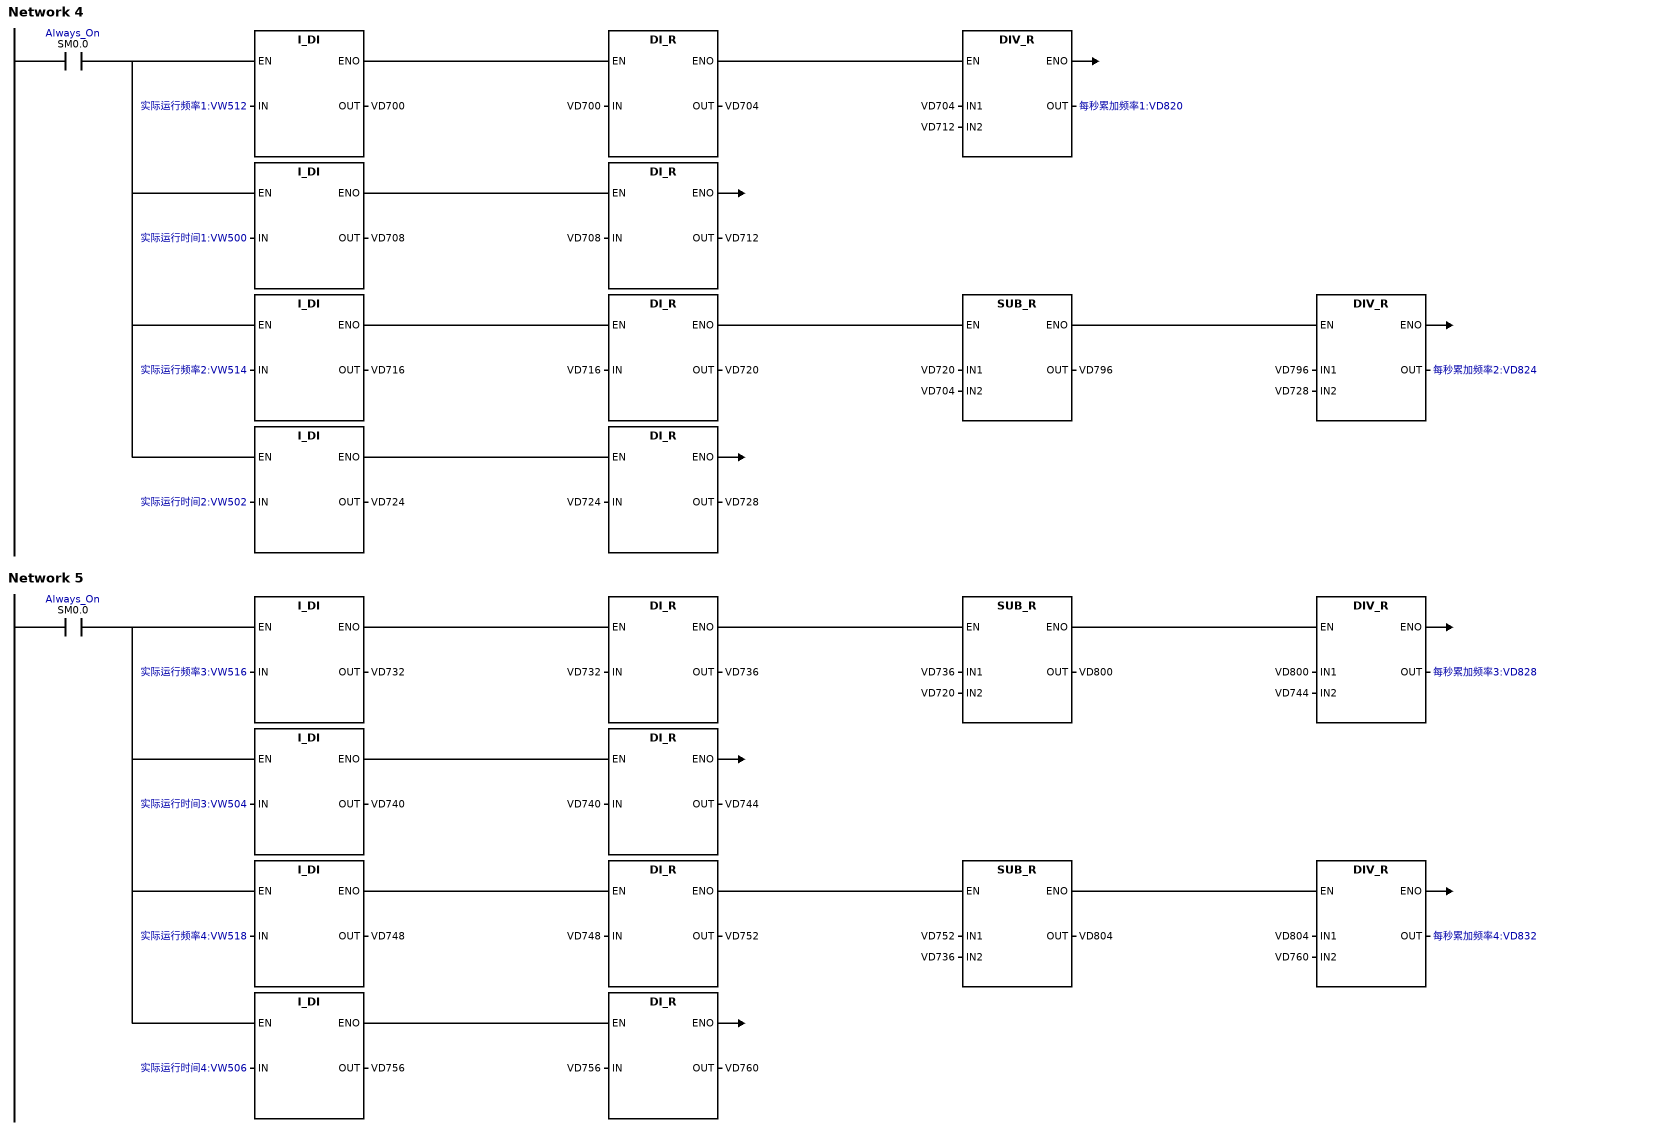
Network 4
LD     Always_On:SM0.0
LPS
ITD    实际运行频率1:VW512, VD700
AENO
DTR    VD700, VD704
AENO
MOVR   VD704, 每秒累加频率1:VD820
/R     VD712, 每秒累加频率1:VD820
LRD
ITD    实际运行时间1:VW500, VD708
AENO
DTR    VD708, VD712
LRD
ITD    实际运行频率2:VW514, VD716
AENO
DTR    VD716, VD720
AENO
MOVR   VD720, VD796
AENO
-R     VD704, VD796
AENO
MOVR   VD796, 每秒累加频率2:VD824
/R     VD728, 每秒累加频率2:VD824
LPP
ITD    实际运行时间2:VW502, VD724
AENO
DTR    VD724, VD728
Network 5
LD     Always_On:SM0.0
LPS
ITD    实际运行频率3:VW516, VD732
AENO
DTR    VD732, VD736
AENO
MOVR   VD736, VD800
AENO
-R     VD720, VD800
AENO
MOVR   VD800, 每秒累加频率3:VD828
/R     VD744, 每秒累加频率3:VD828
LRD
ITD    实际运行时间3:VW504, VD740
AENO
DTR    VD740, VD744
LRD
ITD    实际运行频率4:VW518, VD748
AENO
DTR    VD748, VD752
AENO
MOVR   VD752, VD804
AENO
-R     VD736, VD804
AENO
MOVR   VD804, 每秒累加频率4:VD832
/R     VD760, 每秒累加频率4:VD832
LPP
ITD    实际运行时间4:VW506, VD756
AENO
DTR    VD756, VD760
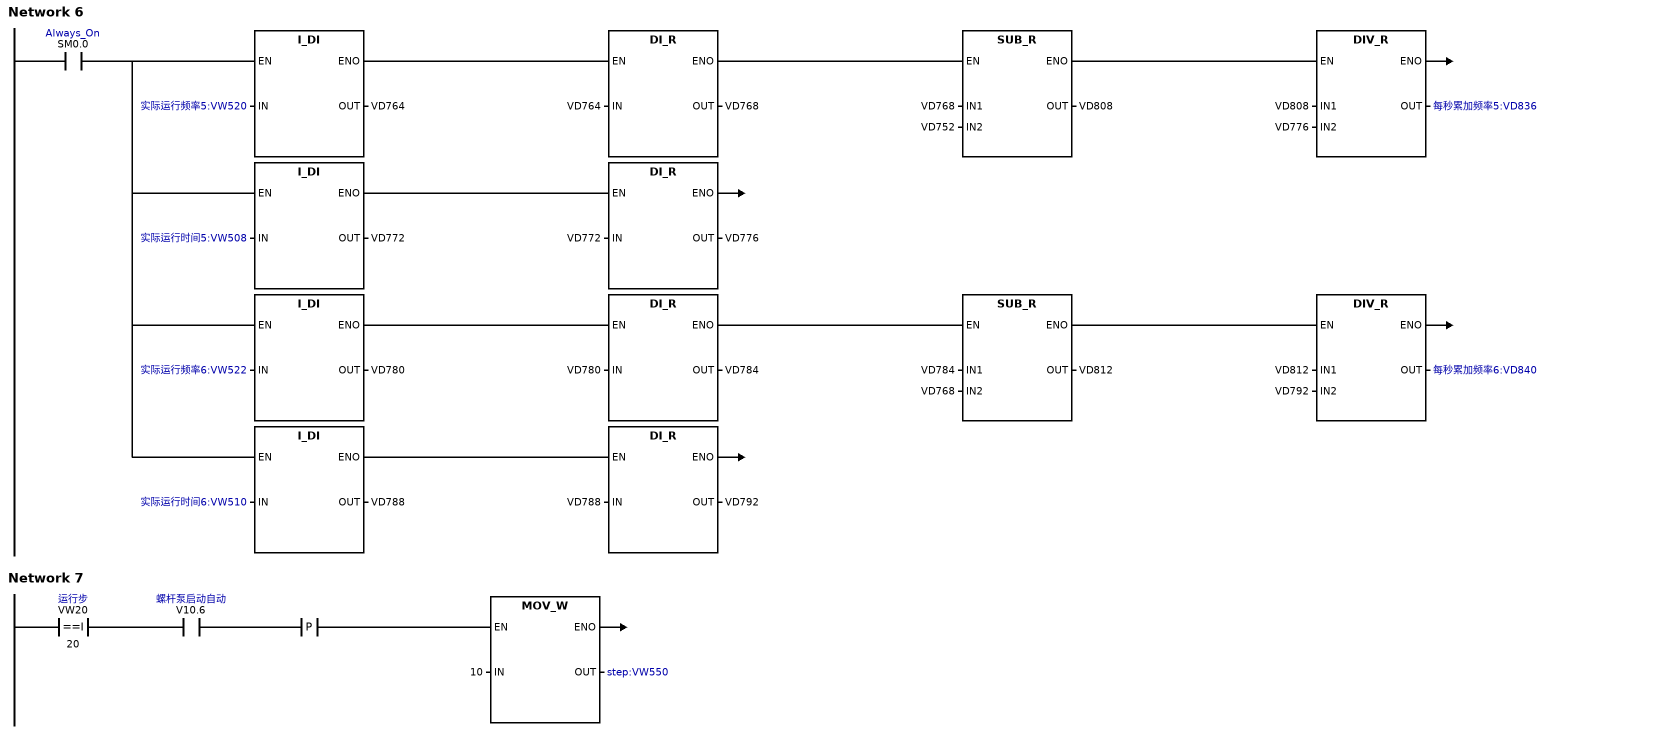
Network 6
LD     Always_On:SM0.0
LPS
ITD    实际运行频率5:VW520, VD764
AENO
DTR    VD764, VD768
AENO
MOVR   VD768, VD808
AENO
-R     VD752, VD808
AENO
MOVR   VD808, 每秒累加频率5:VD836
/R     VD776, 每秒累加频率5:VD836
LRD
ITD    实际运行时间5:VW508, VD772
AENO
DTR    VD772, VD776
LRD
ITD    实际运行频率6:VW522, VD780
AENO
DTR    VD780, VD784
AENO
MOVR   VD784, VD812
AENO
-R     VD768, VD812
AENO
MOVR   VD812, 每秒累加频率6:VD840
/R     VD792, 每秒累加频率6:VD840
LPP
ITD    实际运行时间6:VW510, VD788
AENO
DTR    VD788, VD792
Network 7
LDW=   运行步:VW20, 20
A      螺杆泵启动自动:V10.6
EU
MOVW   10, step:VW550
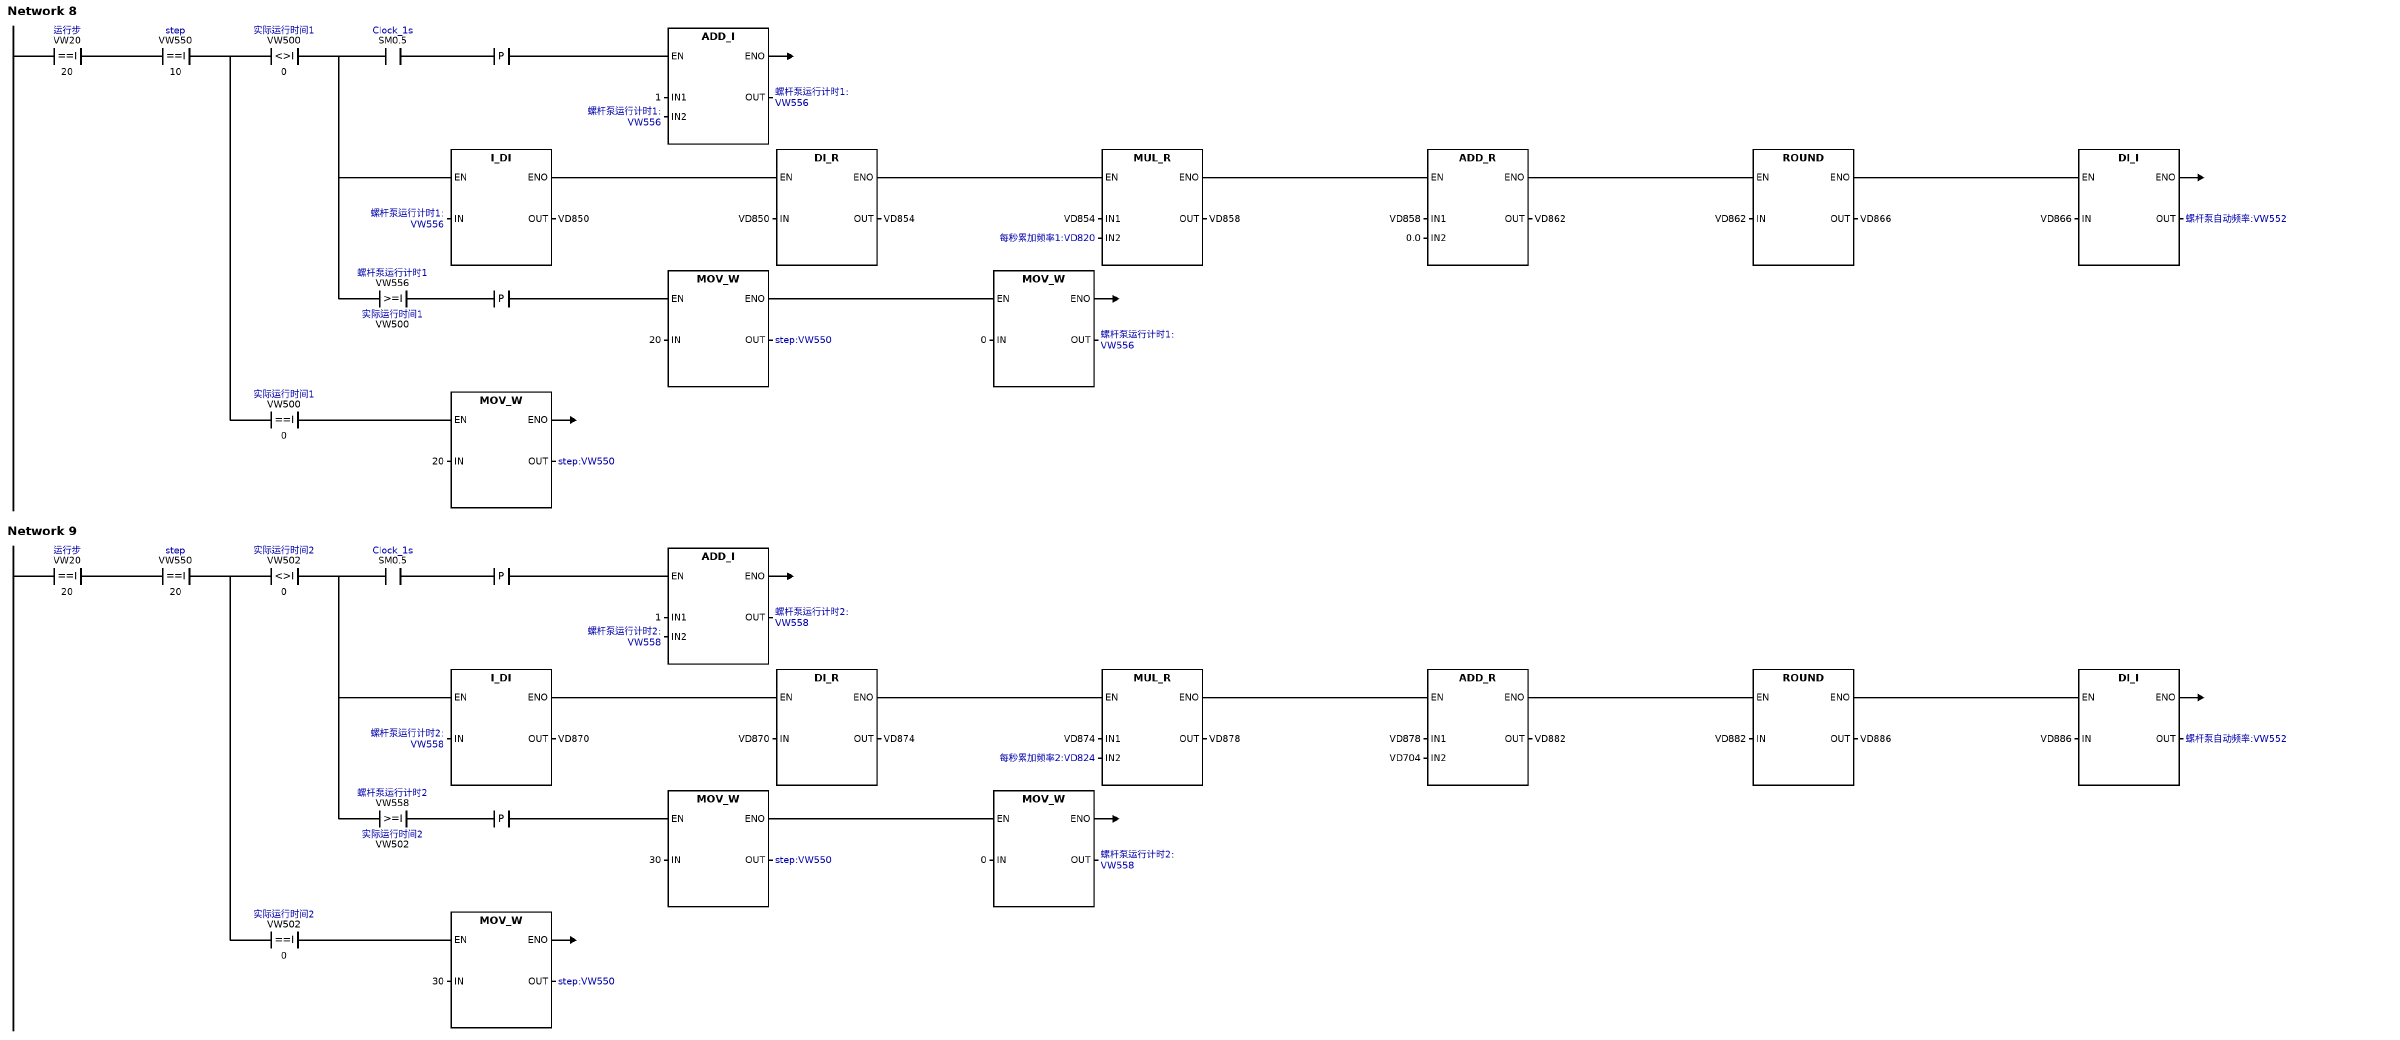
Network 8
LDW=   运行步:VW20, 20
AW=    step:VW550, 10
LPS
AW<>   实际运行时间1:VW500, 0
LPS
A      Clock_1s:SM0.5
EU
+I     1, 螺杆泵运行计时1:VW556
LRD
ITD    螺杆泵运行计时1:VW556, VD850
AENO
DTR    VD850, VD854
AENO
MOVR   VD854, VD858
AENO
*R     每秒累加频率1:VD820, VD858
AENO
MOVR   VD858, VD862
AENO
+R     0.0, VD862
AENO
ROUND  VD862, VD866
AENO
DTI    VD866, 螺杆泵自动频率:VW552
LPP
AW>=   螺杆泵运行计时1:VW556, 实际运行时间1:VW500
EU
MOVW   20, step:VW550
AENO
MOVW   0, 螺杆泵运行计时1:VW556
LPP
AW=    实际运行时间1:VW500, 0
MOVW   20, step:VW550
Network 9
LDW=   运行步:VW20, 20
AW=    step:VW550, 20
LPS
AW<>   实际运行时间2:VW502, 0
LPS
A      Clock_1s:SM0.5
EU
+I     1, 螺杆泵运行计时2:VW558
LRD
ITD    螺杆泵运行计时2:VW558, VD870
AENO
DTR    VD870, VD874
AENO
MOVR   VD874, VD878
AENO
*R     每秒累加频率2:VD824, VD878
AENO
MOVR   VD878, VD882
AENO
+R     VD704, VD882
AENO
ROUND  VD882, VD886
AENO
DTI    VD886, 螺杆泵自动频率:VW552
LPP
AW>=   螺杆泵运行计时2:VW558, 实际运行时间2:VW502
EU
MOVW   30, step:VW550
AENO
MOVW   0, 螺杆泵运行计时2:VW558
LPP
AW=    实际运行时间2:VW502, 0
MOVW   30, step:VW550
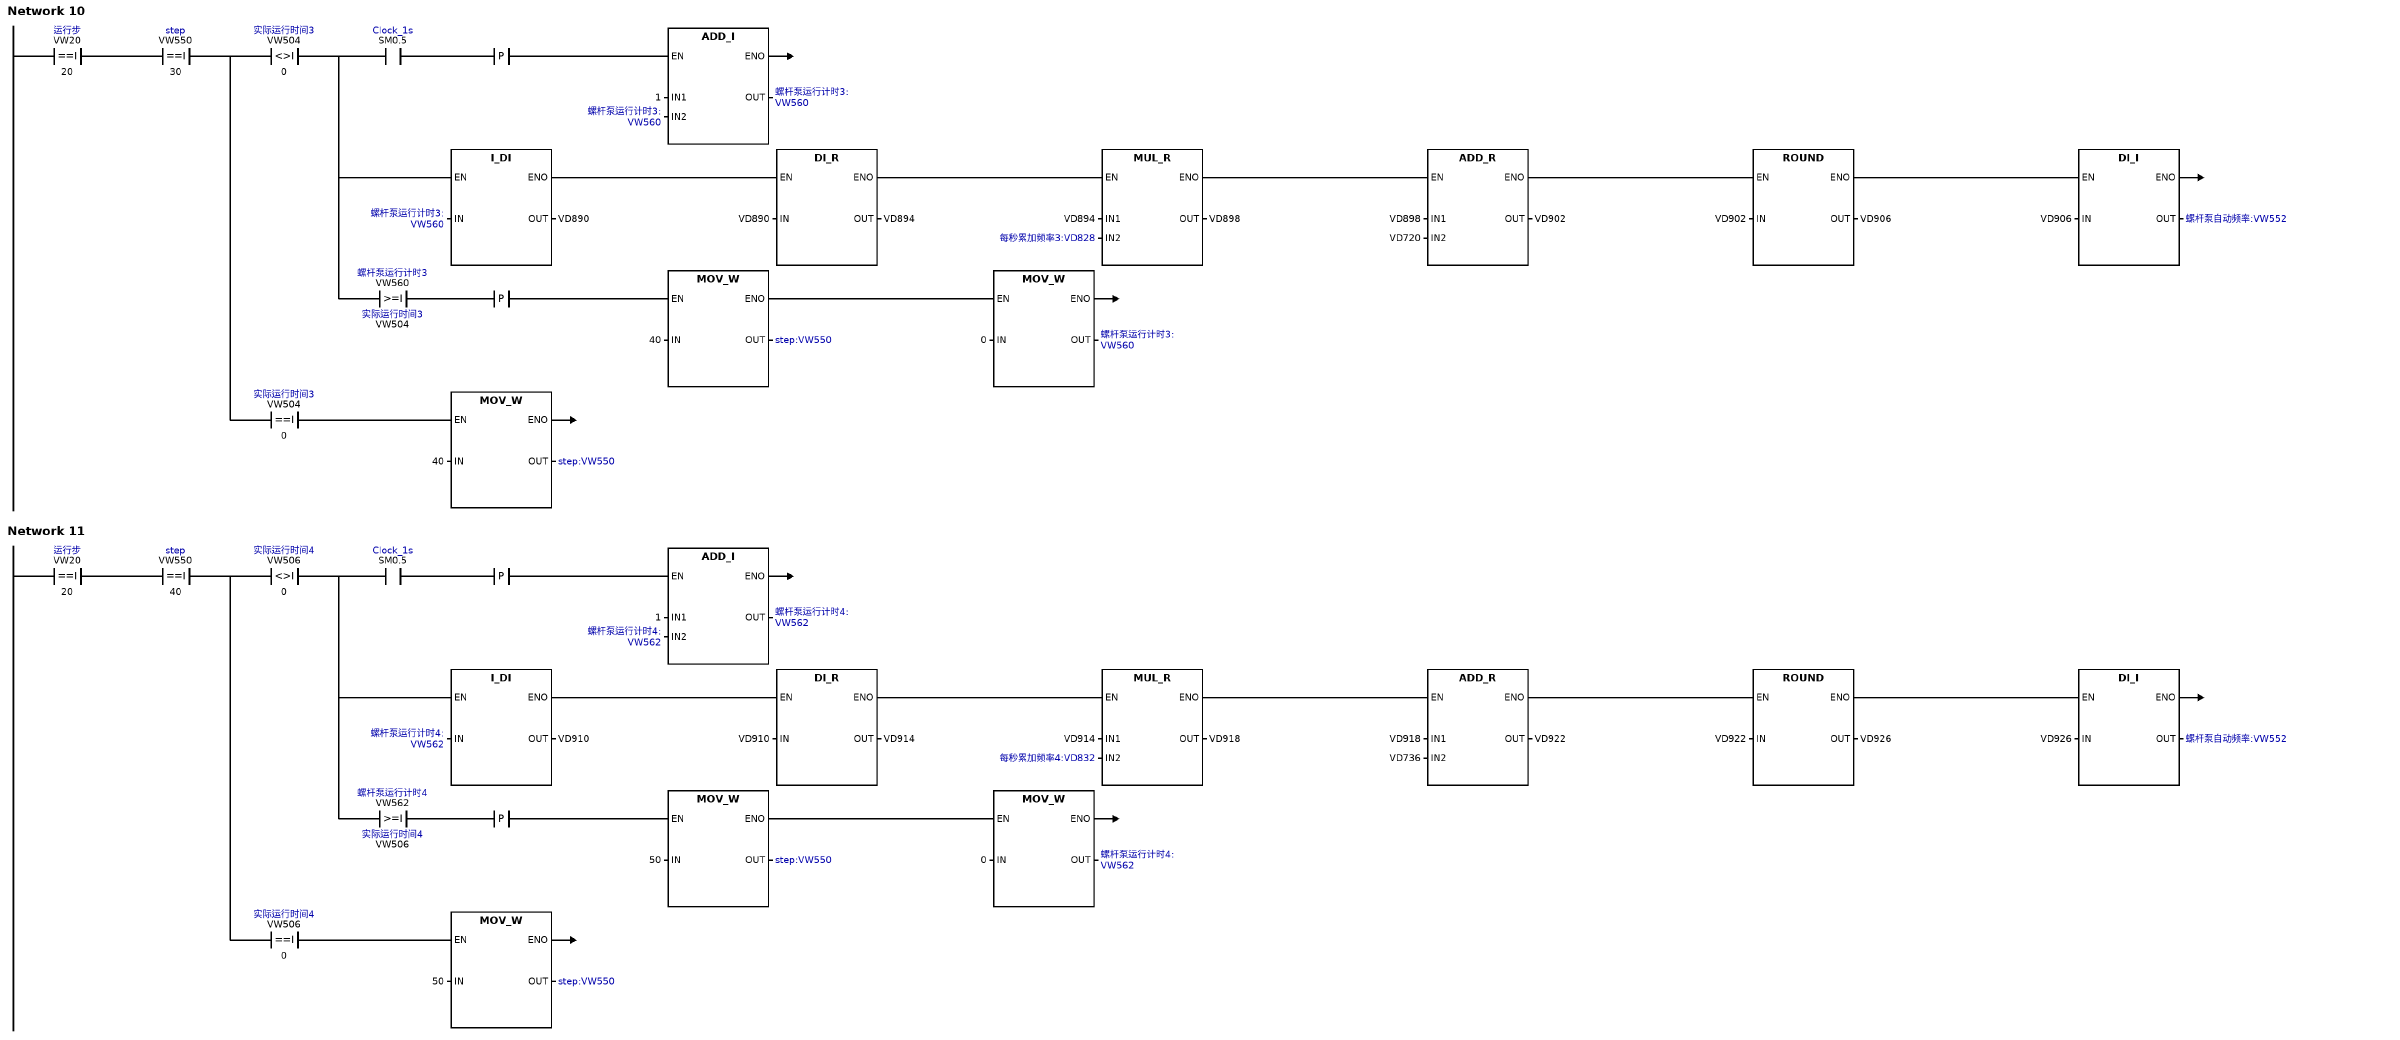
Network 10
LDW=   运行步:VW20, 20
AW=    step:VW550, 30
LPS
AW<>   实际运行时间3:VW504, 0
LPS
A      Clock_1s:SM0.5
EU
+I     1, 螺杆泵运行计时3:VW560
LRD
ITD    螺杆泵运行计时3:VW560, VD890
AENO
DTR    VD890, VD894
AENO
MOVR   VD894, VD898
AENO
*R     每秒累加频率3:VD828, VD898
AENO
MOVR   VD898, VD902
AENO
+R     VD720, VD902
AENO
ROUND  VD902, VD906
AENO
DTI    VD906, 螺杆泵自动频率:VW552
LPP
AW>=   螺杆泵运行计时3:VW560, 实际运行时间3:VW504
EU
MOVW   40, step:VW550
AENO
MOVW   0, 螺杆泵运行计时3:VW560
LPP
AW=    实际运行时间3:VW504, 0
MOVW   40, step:VW550
Network 11
LDW=   运行步:VW20, 20
AW=    step:VW550, 40
LPS
AW<>   实际运行时间4:VW506, 0
LPS
A      Clock_1s:SM0.5
EU
+I     1, 螺杆泵运行计时4:VW562
LRD
ITD    螺杆泵运行计时4:VW562, VD910
AENO
DTR    VD910, VD914
AENO
MOVR   VD914, VD918
AENO
*R     每秒累加频率4:VD832, VD918
AENO
MOVR   VD918, VD922
AENO
+R     VD736, VD922
AENO
ROUND  VD922, VD926
AENO
DTI    VD926, 螺杆泵自动频率:VW552
LPP
AW>=   螺杆泵运行计时4:VW562, 实际运行时间4:VW506
EU
MOVW   50, step:VW550
AENO
MOVW   0, 螺杆泵运行计时4:VW562
LPP
AW=    实际运行时间4:VW506, 0
MOVW   50, step:VW550
